// This function has been automatically generated from the project information.
{attribute 'signature_flag' := '1073741824'}
{attribute 'TcGenerated'}
{attribute 'no-analysis'}
FUNCTION F_GetTitle : WSTRING
VAR_INPUT
	
END_VAR

F_GetTitle := "Event Video Playback";

END_FUNCTION

(* stored: Version 1.1.0.1
   POU F_GetTitle: Id {ce94e1c6-da39-08b9-38b7-1b327f7867f9}, SpecialFunc None *)
